(* CODESYS project TCP Server Example.project

Project tree, tasks and I/O mapping:
  Device : CODESYS Control for Raspberry Pi, 3S - Smart Software Solutions GmbH, version 3.5.11.20
    application Application
      libraries: Standard, * (System); Network, 3.5.7.0 (3S - Smart Software Solutions GmbH); Raspberry I2C Gyroscopes, 1.1.1.0 (3S - Smart Software Solutions GmbH)
      task MainTask (cyclic, interval 4 ms, priority 1) calls PLC_PRG
      task VISU_TASK (cyclic, interval 100 ms, priority 31) calls VisuElems.Visu_Prg
      program PLC_PRG [CFC]
      function block TCPServer [ST]
      visualisation Visualization
    SoftMotion General Axis Pool
    I²C
    SPI
    GPIOs_A_B : GPIOs A/B, 3S - Smart Software Solutions GmbH, version 3.5.11.0
        unmapped channels: digital inputs (GPIO0..GPIO31), digital outputs (GPIO0..GPIO31)
    Onewire
    Camera device
      <Leer>
  text list GlobalTextList
*)

// Device/Application/PLC_PRG
PROGRAM PLC_PRG
VAR
	taster: BOOL;
	TCPServer_0: TCPServer;
END_VAR

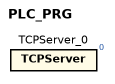
TCPServer_0(); // TCPServer

END_PROGRAM

// Device/Application/TCPServer
FUNCTION_BLOCK TCPServer
VAR_INPUT
END_VAR
VAR_OUTPUT
END_VAR
VAR
	tcpServer: nbs.TCP_Server;
	tcpConnection: nbs.TCP_Connection;
	tcpWrite: nbs.TCP_Write;
	tcpRead: nbs.TCP_Read;
    receivedData : ARRAY [0..255] OF BYTE;
    transmitData : ARRAY [0..255] OF BYTE;
	tempdata: STRING := 'hello';
    startSend : BOOL;
    transmitCount : WORD;
    receiveCount : DINT;
    dataWrite: STRING;
    index: DINT;
    result : BOOL;
	ipAddr: NBS.IP_ADDR;
	data: NBS.CAA.PVOID;
END_VAR


data := ADR(tempdata);

ipAddr.sAddr := '0.0.0.0';
tcpServer(xEnable:=TRUE, uiPort:=4444, ipAddr:=ipAddr);

tcpConnection(xEnable:=TRUE, hServer:=tcpServer.hServer);

IF NOT tcpConnection.xActive THEN
	tcpRead(xEnable:=TRUE, hConnection:=tcpConnection.hConnection, pData:=ADR(receivedData), szSize:=SIZEOF(receivedData));
    //tcpWrite(hConnection:=tcpConnection.hConnection, udiTimeOut:=10000, xExecute:=TRUE, pData:=ADR(data), szSize:=SIZEOF(tempdata));
END_IF

END_FUNCTION_BLOCK

// Device/Application/Visualization
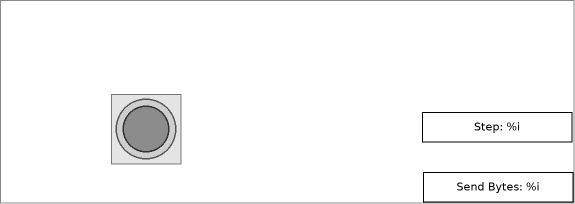
VISUALIZATION Visualization  // 575x204
    PushSwitch (111,94 70x70), variable: PLC_PRG.taster, behaviour: TAP, style: Switch-PushSwitch-Gray
    Rectangle (422,112 150x30), "Step: %i"
    Rectangle (423,172 150x30), "Send Bytes: %i"
END_VISUALIZATION
